(* IEC 61131-3 sources: Industry-PLC-LLM/data/PLCBEAD_repo/PLCBEAD_PLCEmbed-main/PLC-BEAD/Source/GEB/INC2, 1 file *)

(* ---- INC2.ST ---- *)
FUNCTION INC2:INT

	VAR_INPUT
		X :	INT;
		D :	INT;
		L :	INT;
		U :	INT;
	END_VAR

	VAR
		tmp :	INT;
	END_VAR

	tmp := U - L + 1;
	INC2 := (X + D - L + tmp) MOD tmp + L;

END_FUNCTION

PROGRAM program0
	VAR
		X :	INT;
		D :	INT;
		L :	INT;
		U :	INT;
		CEIL5_OUT : INT;
	END_VAR

  	CEIL5_OUT := INC2(X, D, L, U);
END_PROGRAM
